FUNCTION_BLOCK FB_LoadRecipe
VAR_INPUT
	sFileName : STRING(255); // Ex: 'C:\TwinCAT\Recipes\NomeDaReceita.json'
    bExecute  : BOOL;
END_VAR
VAR_OUTPUT
	bBusy   : BOOL;
    bDone   : BOOL;
    bError  : BOOL;
    nErrId  : UDINT;
END_VAR
VAR
	fbFileOpen  : FB_FileOpen;
    fbFileRead  : FB_FileRead;
    fbFileClose : FB_FileClose;
    fbJson      : FB_JsonDomParser;

    hFile    	: UINT;
    sBuffer  	: STRING(16384);
    jsonRoot 	: SJsonValue;
    jsonVal  	: SJsonValue;
	nBytesRead  : UDINT;
    idx      	: INT;
    iStep     	: INT;

    sPath    : STRING(255);
END_VAR

IF NOT bExecute THEN
	bBusy := FALSE;
	bDone := FALSE;
	bError := FALSE;
	nErrId := 0;
	sBuffer := '';
	fbFileOpen(bExecute := FALSE);
	fbFileRead(bExecute := FALSE);
	fbFileClose(bExecute := FALSE);
	iStep := 0;
END_IF


CASE iStep OF
0:
    IF bExecute THEN
        bBusy := TRUE;
        bDone := FALSE;
        bError := FALSE;
        nErrId := 0;

        fbFileOpen(
            sNetId := '',
            sPathName := sFileName,
            nMode := FOPEN_MODEREAD OR FOPEN_MODETEXT,
            bExecute := TRUE
        );
		sBuffer := '';
        iStep := 10;
    END_IF

10:
    fbFileOpen(bExecute := FALSE);
    IF NOT fbFileOpen.bBusy THEN
        IF fbFileOpen.bError THEN
            bError := TRUE;
            nErrId := fbFileOpen.nErrId;
            iStep := 100;
        ELSE
            hFile := fbFileOpen.hFile;
            fbFileRead(
                sNetId := '',
                hFile := hFile,
                pReadBuff := ADR(sBuffer),
                cbReadLen := SIZEOF(sBuffer),
                bExecute := TRUE
            );
            iStep := 20;
        END_IF
    END_IF

20:
    fbFileRead(bExecute := FALSE, sNetId := '', hFile := hFile, pReadBuff := ADR(sBuffer), cbReadLen := SIZEOF(sBuffer), cbRead => nBytesRead);
    IF NOT fbFileRead.bBusy THEN
        IF fbFileRead.bError THEN
            bError := TRUE;
            nErrId := fbFileRead.nErrId;
            iStep := 90;
        ELSE
			// Clear the buffer
            IF nBytesRead < SIZEOF(sBuffer) THEN
    			sBuffer[nBytesRead] := 0; 
			END_IF
            fbFileClose(sNetId := '', hFile := hFile, bExecute := TRUE);
            iStep := 30;
        END_IF
    END_IF

30:
    fbFileClose(bExecute := FALSE);
    IF NOT fbFileClose.bBusy THEN
        IF fbFileClose.bError THEN
            bError := TRUE;
            nErrId := fbFileClose.nErrId;
            iStep := 100;
        ELSE
            iStep := 40;
        END_IF
    END_IF

40:
    jsonRoot := fbJson.ParseDocument(sBuffer);
    IF jsonRoot = 0 THEN
        bError := TRUE;
        nErrId := 16#F1000001; // Código customizado para JSON inválido
        iStep := 100;
    ELSE
        iStep := 50;
    END_IF

50: //Fill the variables with Json buffer info [Parse Json file]
    sPath := 'stInfo/sMethodName';
    GVL_Recipe.stCurrentRecipe.stInfo.sMethodName := fbJson.GetString(fbJson.FindMemberPath(jsonRoot, sPath));

    sPath := 'stInfo/sCreatedBy';
    GVL_Recipe.stCurrentRecipe.stInfo.sCreatedBy := fbJson.GetString(fbJson.FindMemberPath(jsonRoot, sPath));

    sPath := 'stInfo/dCreationDate';
    GVL_Recipe.stCurrentRecipe.stInfo.dCreationDate := STRING_TO_DATE(fbJson.GetString(fbJson.FindMemberPath(jsonRoot, sPath)));

    sPath := 'stInfo/iRevision';
    GVL_Recipe.stCurrentRecipe.stInfo.iRevision := DINT_TO_INT(fbJson.GetInt(fbJson.FindMemberPath(jsonRoot, sPath)));

    FOR idx := 1 TO 4 DO
        sPath := CONCAT('stSolventsTimes/aSolventN#', INT_TO_STRING(idx-1));
        GVL_Recipe.stCurrentRecipe.stSolventsTimes.aSolventN[idx] := TO_USINT(fbJson.GetInt(fbJson.FindMemberPath(jsonRoot, sPath)));

        sPath := CONCAT('stSolventsTimes/aTime#', INT_TO_STRING(idx-1));
        GVL_Recipe.stCurrentRecipe.stSolventsTimes.aTime[idx] := STRING_TO_TIME(fbJson.GetString(fbJson.FindMemberPath(jsonRoot, sPath)));

        sPath := CONCAT('stSolventsTimes/aVelocity#', INT_TO_STRING(idx-1));
        GVL_Recipe.stCurrentRecipe.stSolventsTimes.aVelocity[idx] := TO_INT(fbJson.GetInt(fbJson.FindMemberPath(jsonRoot, sPath)));
    END_FOR

    FOR idx := 1 TO 4 DO
        sPath := CONCAT('stVolumes/aT_IC_Volume#', INT_TO_STRING(idx-1));
        GVL_Recipe.stCurrentRecipe.stVolumes.aT_IC_Volume[idx] := LREAL_TO_REAL(fbJson.GetDouble(fbJson.FindMemberPath(jsonRoot, sPath)));
		
		sPath := CONCAT('stVolumes/aS0_Volume#', INT_TO_STRING(idx-1));
        GVL_Recipe.stCurrentRecipe.stVolumes.aS0_Volume[idx] := LREAL_TO_REAL(fbJson.GetDouble(fbJson.FindMemberPath(jsonRoot, sPath)));
		
		sPath := CONCAT('stVolumes/aS1_Volume#', INT_TO_STRING(idx-1));
        GVL_Recipe.stCurrentRecipe.stVolumes.aS1_Volume[idx] := LREAL_TO_REAL(fbJson.GetDouble(fbJson.FindMemberPath(jsonRoot, sPath)));
		
		sPath := CONCAT('stVolumes/aS2_Volume#', INT_TO_STRING(idx-1));
        GVL_Recipe.stCurrentRecipe.stVolumes.aS2_Volume[idx] := LREAL_TO_REAL(fbJson.GetDouble(fbJson.FindMemberPath(jsonRoot, sPath)));
		
		sPath := CONCAT('stVolumes/aS3_Volume#', INT_TO_STRING(idx-1));
        GVL_Recipe.stCurrentRecipe.stVolumes.aS3_Volume[idx] := LREAL_TO_REAL(fbJson.GetDouble(fbJson.FindMemberPath(jsonRoot, sPath)));
		
		sPath := CONCAT('stVolumes/aS4_Volume#', INT_TO_STRING(idx-1));
        GVL_Recipe.stCurrentRecipe.stVolumes.aS4_Volume[idx] := LREAL_TO_REAL(fbJson.GetDouble(fbJson.FindMemberPath(jsonRoot, sPath)));
		
		sPath := CONCAT('stVolumes/aS5_Volume#', INT_TO_STRING(idx-1));
        GVL_Recipe.stCurrentRecipe.stVolumes.aS5_Volume[idx] := LREAL_TO_REAL(fbJson.GetDouble(fbJson.FindMemberPath(jsonRoot, sPath)));
		
		sPath := CONCAT('stVolumes/aS6_Volume#', INT_TO_STRING(idx-1));
        GVL_Recipe.stCurrentRecipe.stVolumes.aS6_Volume[idx] := LREAL_TO_REAL(fbJson.GetDouble(fbJson.FindMemberPath(jsonRoot, sPath)));
		
		sPath := CONCAT('stVolumes/aS7_Volume#', INT_TO_STRING(idx-1));
        GVL_Recipe.stCurrentRecipe.stVolumes.aS7_Volume[idx] := LREAL_TO_REAL(fbJson.GetDouble(fbJson.FindMemberPath(jsonRoot, sPath)));
		
		sPath := CONCAT('stVolumes/aF_Volume#', INT_TO_STRING(idx-1));
        GVL_Recipe.stCurrentRecipe.stVolumes.aF_Volume[idx] := LREAL_TO_REAL(fbJson.GetDouble(fbJson.FindMemberPath(jsonRoot, sPath)));
		
    END_FOR

    sPath := 'stOtherParams/tSoakTime';
    GVL_Recipe.stCurrentRecipe.stOtherParams.tSoakTime := STRING_TO_TIME(fbJson.GetString(fbJson.FindMemberPath(jsonRoot, sPath)));
	
	sPath := 'stOtherParams/tAgitate1Time';
    GVL_Recipe.stCurrentRecipe.stOtherParams.tAgitate1Time := STRING_TO_TIME(fbJson.GetString(fbJson.FindMemberPath(jsonRoot, sPath)));
	
	sPath := 'stOtherParams/tAgitate2Time';
    GVL_Recipe.stCurrentRecipe.stOtherParams.tAgitate2Time := STRING_TO_TIME(fbJson.GetString(fbJson.FindMemberPath(jsonRoot, sPath)));
	
	sPath := 'stOtherParams/iVialsToFill';
    GVL_Recipe.stCurrentRecipe.stOtherParams.iVialsToFill := TO_USINT(fbJson.GetInt(fbJson.FindMemberPath(jsonRoot, sPath)));
	
	sPath := 'stOtherParams/rVialPrimeVol';
    GVL_Recipe.stCurrentRecipe.stOtherParams.rVialPrimeVol := LREAL_TO_REAL(fbJson.GetDouble(fbJson.FindMemberPath(jsonRoot, sPath)));
	
	sPath := 'stOtherParams/rVial1FillVol';
    GVL_Recipe.stCurrentRecipe.stOtherParams.rVial1FillVol := LREAL_TO_REAL(fbJson.GetDouble(fbJson.FindMemberPath(jsonRoot, sPath)));
	
	sPath := 'stOtherParams/rVials2_4FillVol';
    GVL_Recipe.stCurrentRecipe.stOtherParams.rVials2_4FillVol := LREAL_TO_REAL(fbJson.GetDouble(fbJson.FindMemberPath(jsonRoot, sPath)));
	
	sPath := 'stOtherParams/tAirDryTime';
    GVL_Recipe.stCurrentRecipe.stOtherParams.tAirDryTime := STRING_TO_TIME(fbJson.GetString(fbJson.FindMemberPath(jsonRoot, sPath)));

    iStep := 60;
	
60: // Fill the HMI datagrids for recipe screen
	//Recipe Header info
	GVL_HMI.stRecipeInfo.sMethodName := GVL_Recipe.stCurrentRecipe.stInfo.sMethodName;
	GVL_HMI.stRecipeInfo.sCreatedBy := GVL_Recipe.stCurrentRecipe.stInfo.sCreatedBy;
	GVL_HMI.stRecipeInfo.dCreationDate := GVL_Recipe.stCurrentRecipe.stInfo.dCreationDate;
	GVL_HMI.stRecipeInfo.iRevision := GVL_Recipe.stCurrentRecipe.stInfo.iRevision;
	
	// Solvents and Times datagrid
	// Row 1: Solvent #
	GVL_HMI.aSolventAndTimesRows[1].Rinse1 := GVL_Recipe.stCurrentRecipe.stSolventsTimes.aSolventN[1];
	GVL_HMI.aSolventAndTimesRows[1].Rinse2 := GVL_Recipe.stCurrentRecipe.stSolventsTimes.aSolventN[2];
	GVL_HMI.aSolventAndTimesRows[1].Wash1  := GVL_Recipe.stCurrentRecipe.stSolventsTimes.aSolventN[3];
	GVL_HMI.aSolventAndTimesRows[1].Wash2  := GVL_Recipe.stCurrentRecipe.stSolventsTimes.aSolventN[4];
	
	// Row 2: Time (seconds)
	GVL_HMI.aSolventAndTimesRows[2].Rinse1 := DWORD_TO_INT(TIME_TO_DWORD(GVL_Recipe.stCurrentRecipe.stSolventsTimes.aTime[1]) / 1000); // TIME in seconds
	GVL_HMI.aSolventAndTimesRows[2].Rinse2 := DWORD_TO_INT(TIME_TO_DWORD(GVL_Recipe.stCurrentRecipe.stSolventsTimes.aTime[2]) / 1000); // TIME in seconds
	GVL_HMI.aSolventAndTimesRows[2].Wash1  := DWORD_TO_INT(TIME_TO_DWORD(GVL_Recipe.stCurrentRecipe.stSolventsTimes.aTime[3]) / 1000); // TIME in seconds
	GVL_HMI.aSolventAndTimesRows[2].Wash2  := DWORD_TO_INT(TIME_TO_DWORD(GVL_Recipe.stCurrentRecipe.stSolventsTimes.aTime[4]) / 1000); // TIME in seconds
	
	// Row 3: Velocity
	GVL_HMI.aSolventAndTimesRows[3].Rinse1 := GVL_Recipe.stCurrentRecipe.stSolventsTimes.aVelocity[1];
	GVL_HMI.aSolventAndTimesRows[3].Rinse2 := GVL_Recipe.stCurrentRecipe.stSolventsTimes.aVelocity[2];
	GVL_HMI.aSolventAndTimesRows[3].Wash1  := GVL_Recipe.stCurrentRecipe.stSolventsTimes.aVelocity[3];
	GVL_HMI.aSolventAndTimesRows[3].Wash2  := GVL_Recipe.stCurrentRecipe.stSolventsTimes.aVelocity[4];
	
	//Volumes Datagrid
	// 1:Rinse1, 2:Rinse2, 3:Wash1, 4:Wash2
    GVL_HMI.aVolumeRows[1].Rinse1 := GVL_Recipe.stCurrentRecipe.stVolumes.aT_IC_Volume[1];
    GVL_HMI.aVolumeRows[1].Rinse2 := GVL_Recipe.stCurrentRecipe.stVolumes.aT_IC_Volume[2];
    GVL_HMI.aVolumeRows[1].Wash1  := GVL_Recipe.stCurrentRecipe.stVolumes.aT_IC_Volume[3];
    GVL_HMI.aVolumeRows[1].Wash2  := GVL_Recipe.stCurrentRecipe.stVolumes.aT_IC_Volume[4];

    GVL_HMI.aVolumeRows[2].Rinse1 := GVL_Recipe.stCurrentRecipe.stVolumes.aS0_Volume[1];
    GVL_HMI.aVolumeRows[2].Rinse2 := GVL_Recipe.stCurrentRecipe.stVolumes.aS0_Volume[2];
    GVL_HMI.aVolumeRows[2].Wash1  := GVL_Recipe.stCurrentRecipe.stVolumes.aS0_Volume[3];
    GVL_HMI.aVolumeRows[2].Wash2  := GVL_Recipe.stCurrentRecipe.stVolumes.aS0_Volume[4];

    GVL_HMI.aVolumeRows[3].Rinse1 := GVL_Recipe.stCurrentRecipe.stVolumes.aS1_Volume[1];
    GVL_HMI.aVolumeRows[3].Rinse2 := GVL_Recipe.stCurrentRecipe.stVolumes.aS1_Volume[2];
   	GVL_HMI.aVolumeRows[3].Wash1  := GVL_Recipe.stCurrentRecipe.stVolumes.aS1_Volume[3];
    GVL_HMI.aVolumeRows[3].Wash2  := GVL_Recipe.stCurrentRecipe.stVolumes.aS1_Volume[4];
	
	GVL_HMI.aVolumeRows[4].Rinse1 := GVL_Recipe.stCurrentRecipe.stVolumes.aS2_Volume[1];
    GVL_HMI.aVolumeRows[4].Rinse2 := GVL_Recipe.stCurrentRecipe.stVolumes.aS2_Volume[2];
   	GVL_HMI.aVolumeRows[4].Wash1  := GVL_Recipe.stCurrentRecipe.stVolumes.aS2_Volume[3];
    GVL_HMI.aVolumeRows[4].Wash2  := GVL_Recipe.stCurrentRecipe.stVolumes.aS2_Volume[4];
	
	GVL_HMI.aVolumeRows[5].Rinse1 := GVL_Recipe.stCurrentRecipe.stVolumes.aS3_Volume[1];
    GVL_HMI.aVolumeRows[5].Rinse2 := GVL_Recipe.stCurrentRecipe.stVolumes.aS3_Volume[2];
   	GVL_HMI.aVolumeRows[5].Wash1  := GVL_Recipe.stCurrentRecipe.stVolumes.aS3_Volume[3];
    GVL_HMI.aVolumeRows[5].Wash2  := GVL_Recipe.stCurrentRecipe.stVolumes.aS3_Volume[4];
	
	GVL_HMI.aVolumeRows[6].Rinse1 := GVL_Recipe.stCurrentRecipe.stVolumes.aS4_Volume[1];
    GVL_HMI.aVolumeRows[6].Rinse2 := GVL_Recipe.stCurrentRecipe.stVolumes.aS4_Volume[2];
   	GVL_HMI.aVolumeRows[6].Wash1  := GVL_Recipe.stCurrentRecipe.stVolumes.aS4_Volume[3];
    GVL_HMI.aVolumeRows[6].Wash2  := GVL_Recipe.stCurrentRecipe.stVolumes.aS4_Volume[4];
	
	GVL_HMI.aVolumeRows[7].Rinse1 := GVL_Recipe.stCurrentRecipe.stVolumes.aS5_Volume[1];
    GVL_HMI.aVolumeRows[7].Rinse2 := GVL_Recipe.stCurrentRecipe.stVolumes.aS5_Volume[2];
   	GVL_HMI.aVolumeRows[7].Wash1  := GVL_Recipe.stCurrentRecipe.stVolumes.aS5_Volume[3];
    GVL_HMI.aVolumeRows[7].Wash2  := GVL_Recipe.stCurrentRecipe.stVolumes.aS5_Volume[4];
	
	GVL_HMI.aVolumeRows[8].Rinse1 := GVL_Recipe.stCurrentRecipe.stVolumes.aS6_Volume[1];
    GVL_HMI.aVolumeRows[8].Rinse2 := GVL_Recipe.stCurrentRecipe.stVolumes.aS6_Volume[2];
   	GVL_HMI.aVolumeRows[8].Wash1  := GVL_Recipe.stCurrentRecipe.stVolumes.aS6_Volume[3];
    GVL_HMI.aVolumeRows[8].Wash2  := GVL_Recipe.stCurrentRecipe.stVolumes.aS6_Volume[4];
	
	GVL_HMI.aVolumeRows[9].Rinse1 := GVL_Recipe.stCurrentRecipe.stVolumes.aS7_Volume[1];
    GVL_HMI.aVolumeRows[9].Rinse2 := GVL_Recipe.stCurrentRecipe.stVolumes.aS7_Volume[2];
   	GVL_HMI.aVolumeRows[9].Wash1  := GVL_Recipe.stCurrentRecipe.stVolumes.aS7_Volume[3];
    GVL_HMI.aVolumeRows[9].Wash2  := GVL_Recipe.stCurrentRecipe.stVolumes.aS7_Volume[4];

    GVL_HMI.aVolumeRows[10].Rinse1 := GVL_Recipe.stCurrentRecipe.stVolumes.aF_Volume[1];
    GVL_HMI.aVolumeRows[10].Rinse2 := GVL_Recipe.stCurrentRecipe.stVolumes.aF_Volume[2];
    GVL_HMI.aVolumeRows[10].Wash1  := GVL_Recipe.stCurrentRecipe.stVolumes.aF_Volume[3];
    GVL_HMI.aVolumeRows[10].Wash2  := GVL_Recipe.stCurrentRecipe.stVolumes.aF_Volume[4];
	
	//Other Params datagrid
	GVL_HMI.aOtherParamsRows[1].Value     := TIME_TO_DWORD(GVL_Recipe.stCurrentRecipe.stOtherParams.tSoakTime) / 1000.0; // Soak Time
	GVL_HMI.aOtherParamsRows[2].Value     := TIME_TO_DWORD(GVL_Recipe.stCurrentRecipe.stOtherParams.tAgitate1Time) / 1000.0; // Agitate 1 Time
	GVL_HMI.aOtherParamsRows[3].Value     := TIME_TO_DWORD(GVL_Recipe.stCurrentRecipe.stOtherParams.tAgitate2Time) / 1000.0; // Agitate 2 Time
	GVL_HMI.aOtherParamsRows[4].Value     := GVL_Recipe.stCurrentRecipe.stOtherParams.iVialsToFill; // Vials to Fill
	GVL_HMI.aOtherParamsRows[5].Value     := GVL_Recipe.stCurrentRecipe.stOtherParams.rVialPrimeVol; // Vial Prime Vol
	GVL_HMI.aOtherParamsRows[6].Value     := GVL_Recipe.stCurrentRecipe.stOtherParams.rVial1FillVol; // Vial 1 Fill Vol
	GVL_HMI.aOtherParamsRows[7].Value     := GVL_Recipe.stCurrentRecipe.stOtherParams.rVials2_4FillVol; // Vials 2-4 Fill Vol
	GVL_HMI.aOtherParamsRows[8].Value     := TIME_TO_DWORD(GVL_Recipe.stCurrentRecipe.stOtherParams.tAirDryTime) / 1000.0; // Air Dry Time
	
	iStep := 100;

90:
    fbFileClose(sNetId := '', hFile := hFile, bExecute := TRUE);
    iStep := 100;
	
100:
    bBusy := FALSE;
    bDone := NOT bError;
    IF NOT bExecute THEN
        iStep := 0;
    END_IF
END_CASE

END_FUNCTION_BLOCK

(* stored: Version 1.1.0.1, ProductVersion 3.1.4024.15
   POU FB_LoadRecipe: Id {fdbedb76-49e0-47f1-8b40-c95081ed8fdc}, SpecialFunc None *)
